(* Logix 5000 project; controller Empty vendor 1 type 14 code 226 rev 34.11; software revision 34.01 *)

TASK Fast (periodic, rate 100 ms, priority 1, watchdog 150 ms) : FastProgram
TASK loop (continuous, watchdog 1000 ms) : MainProgram
TASK Normal (periodic, rate 250 ms, priority 2, watchdog 375 ms) : NormalProgram
TASK SafetyTask (periodic, rate 20 ms, priority 10, watchdog 20 ms, safety) : SafetyProgram
TASK Slow (periodic, rate 500 ms, priority 3, watchdog 750 ms) : SlowProgram
TASK System (periodic, rate 1000 ms, priority 4, watchdog 1500 ms) : SystemProgram

MODULES
   Local : vendor 1 type 14 code 226 (5069 0, rev 34.11)
END_MODULES

ADD_ON_INSTRUCTION GradientSearchMin   (* revision 1.0 *)
VAR_INPUT
   x01 : LREAL; {access None, required}
   x02 : LREAL; {access None, required}
   iter : INT; {access None, required}
END_VAR
VAR_OUTPUT
   GradientSearchMin1 : LREAL; {access None, required}
END_VAR
VAR
   x1 : LREAL; {access None}
   x2 : LREAL; {access None}
   delta : LREAL; {access None}
   alpha : LREAL; {access None}
   y : LREAL; {access None}
   y1 : LREAL; {access None}
   y2 : LREAL; {access None}
   dy_dx1 : LREAL; {access None}
   dy_dx2 : LREAL; {access None}
   OF_tmp : OptimizedFunction; {access None}
   x1_delta : LREAL; {access None}
   x2_delta : LREAL; {access None}
END_VAR

ROUTINE Logic   (* structured text *)
   
   delta := 0.001;
   alpha := 1.0;
   
   x1 := x01;
   x2 := x02;
   
   WHILE iter >= 0 DO
       iter := iter - 1;
   
       // calculate gradient
   	x1_delta := x1 + delta;
   	x2_delta := x2 + delta;
       OptimizedFunction(OF_tmp, x1, x2, y);
       OptimizedFunction(OF_tmp, x1_delta, x2, y1);
       OptimizedFunction(OF_tmp, x1, x2_delta, y2);
   
       dy_dx1 := (y1 - y) / delta;
       dy_dx2 := (y2 - y) / delta;
   
       x1 := x1 - alpha * dy_dx1;
       x2 := x2 - alpha * dy_dx2;
   
   END_WHILE;
   
   OptimizedFunction(OF_tmp,x1, x2,GradientSearchMin1);
   
   // OptimizedFunction(OF_tmp,x1,x2,GradientSearchMin1);
   
   
   
   
END_ROUTINE
END_ADD_ON_INSTRUCTION

ADD_ON_INSTRUCTION OptimizedFunction   (* revision 1.0 *)
VAR_INPUT
   x1 : LREAL; {required}
   x2 : LREAL; {required}
END_VAR
VAR_OUTPUT
   OptimizedFunction1 : LREAL; {required}
END_VAR

ROUTINE Logic   (* structured text *)
   
   OptimizedFunction1 := x1 ** 2.0
   - 6.0 * x1 ** 2.0 * x2 - 20.0 * x1 + 3.0 * x2 ** 2.0 + 3.0 * x1 ** 4.0 + 109.0;
   
   
END_ROUTINE
END_ADD_ON_INSTRUCTION

PROGRAM FastProgram   (* main routine MainRoutine *)

ROUTINE MainRoutine   (* ladder *)
END_ROUTINE
END_PROGRAM

PROGRAM MainProgram   (* main routine main *)
VAR
   gsm_tmp : GradientSearchMin;
   minimum : LREAL;
END_VAR

ROUTINE main   (* structured text *)
   
   
   
   
   
   GradientSearchMin(gsm_tmp, 100.0, 100.0, 1000, minimum);
   
   
END_ROUTINE
END_PROGRAM

PROGRAM NormalProgram   (* main routine MainRoutine *)

ROUTINE MainRoutine   (* ladder *)
END_ROUTINE
END_PROGRAM

PROGRAM SafetyProgram   (* main routine MainRoutine, safety *)

ROUTINE MainRoutine   (* ladder *)
END_ROUTINE
END_PROGRAM

PROGRAM SlowProgram   (* main routine MainRoutine *)

ROUTINE MainRoutine   (* ladder *)
END_ROUTINE
END_PROGRAM

PROGRAM SystemProgram   (* main routine MainRoutine *)

ROUTINE MainRoutine   (* ladder *)
END_ROUTINE
END_PROGRAM
